FUNCTION_BLOCK ClearLinkEIP
VAR_INPUT
	bEnable : BOOL;
END_VAR
VAR_OUTPUT
	pulse AT %Q* : INT; //num pulses
	outputRegister AT %Q* : INT;
	brakeRelease AT %Q* : BOOL;
	
	A : BOOL; //direction (F = inwards, T = outwards)
	B : BOOL; //home bit
	clear : BOOL;
	
	contact AT %I* : BOOL;
	home AT %I* : BOOL;
	outerLimit AT %I* : BOOL;
	innerLimit AT %I* : BOOL;
	
	hlfb AT %I* : REAL; //high level feedback, if -9999 then servo is idle
	
	homeSet : BOOL;
	busy : BOOL;
	error : BOOL;
	
	position : LREAL;
	targetPos : LREAL;
END_VAR
VAR
	pulseRequest : INT;
	pulser : TON;
	
	minHoming : TON;
	resetPulse : TP;
	
	step : Homing;
	mode : (DISABLE, HOLD, TARGET, CONTINUOUS, RESET_ERR);
END_VAR
VAR_STAT CONSTANT
	resetTime : TIME := T#1000MS;
	pulseWidth : TIME := T#40MS;
	pulseSeparation : TIME := T#40MS;
	unitsPerPulse : INT := 800; //800 Teknic units per revolution
	distancePerPulse : INT := 5; //5mm per revolution
END_VAR

//M-connector output register
outputRegister.0 := bEnable; 	//enable
outputRegister.1 := A; 			//direction bit
outputRegister.2 := B; 			//homing bit - set to TRUE on startup to begin homing, then set to FALSE to finish homing
outputRegister.3 := clear; 		//reset bit

resetPulse(IN:= , PT:= resetTime, Q=> clear, ET=> ); //reset timer

IF NOT bEnable THEN
	homeSet := FALSE;
	mode := HOLD;
END_IF

//set the bool outputs, all are listed for readability
homeSet := homeSet;
busy := hlfb <> -9999;
error := error;

override(); //if sensor limits are reached, this method blocks motion that would exceed the limits

CASE mode OF		
	HOLD: //hold current position, no motion
		pulse := 0;
		pulseRequest := 0;
	
	TARGET:	//target a given position
		IF WithinTolerance(position, targetPos, distancePerPulse) THEN
			pulseRequest := 0;
			mode := HOLD;
			
		ELSIF NOT busy THEN
			A :=  position < targetPos;
			(*
			2 options to traverse to a target position:
				a)  send all pulses at once - single continuous motion but may exceed limits
				b)  1 pulse at a time - choppy but safer
			*)
			pulseRequest := TO_INT(ABS(position - targetPos)/distancePerPulse);
			//pulseRequest := 1;
			
		END_IF
		
	CONTINUOUS: //single pulses in the direction specified by moveContinuous()
		pulseRequest := 1;
		
	RESET_ERR: //reset pulse
		pulse := 0;
		pulseRequest := 0;
		
		resetPulse.IN := TRUE;
		mode := HOLD;
		(*
		IF resetTimer.Q THEN
			resetTimer.IN := FALSE;
			mode := HOLD;
		END_IF
		*)
		
END_CASE

sequence();

METHOD homingSequence : BOOL
minHoming(IN:= , PT:= T#1S, Q=> , ET=> ); //IN and OUT should be held for at least 1 second - may be removed for deployment

IF NOT bEnable THEN //homing does not begin until software enable
	RETURN;
END_IF

CASE step OF
	Homing.IDLE:
		bEnable := FALSE;
		A := FALSE;
		B := FALSE;
		brakeRelease := TRUE;
		
		homeSet := FALSE;
		step := Homing.IN;
		
	Homing.IN: //let insertion drop to inner limit before homing
		bEnable := FALSE;
		A := FALSE;
		B := FALSE;
		brakeRelease := TRUE;
		
		minHoming.IN := TRUE;
		
		IF NOT innerLimit AND minHoming.Q THEN
			minHoming.IN := FALSE;
			step := Homing.OUT;
		END_IF
	
	Homing.OUT: //home to outer limit
		bEnable := TRUE;
		A := FALSE;
		B := TRUE;
		brakeRelease := TRUE;
		
		minHoming.IN := TRUE;
		
		IF NOT home AND minHoming.Q THEN
			minHoming.IN := FALSE;
			step := Homing.DONE;
		END_IF
		
	Homing.DONE: //set home
		bEnable := TRUE;
		A := FALSE;
		B := FALSE;
		brakeRelease := TRUE;
		
		position := 0;
		
		homeSet := TRUE;
		homingSequence := TRUE;
		
		mode := HOLD;
		step := Homing.IDLE;
		
END_CASE
END_METHOD

METHOD moveAbsolute : BOOL
VAR_INPUT
	newTarget : LREAL;
END_VAR
targetPos := newTarget;
mode := TARGET;
END_METHOD

METHOD moveContinuous : BOOL
VAR_INPUT
	direction : MC_Direction;
END_VAR
IF direction = MC_Negative_Direction THEN
	A := FALSE;
ELSIF direction = MC_Positive_Direction THEN
	A := TRUE;
END_IF

mode := CONTINUOUS;
END_METHOD

METHOD PRIVATE override : BOOL
VAR_INPUT
END_VAR
(*
IF (*NOT*) home THEN //block outwards motion
	position := 0;
	IF A THEN
		mode := HOLD;
	END_IF
	
ELSIF (*NOT*) outerLimit AND_THEN A THEN //block outwards motion
	mode := HOLD;

ELSIF (*NOT*) innerLimit AND_THEN NOT A THEN //block inwards motion
	mode := HOLD;
	
END_IF
*)


IF
	((*NOT*) home AND_THEN A) OR
	((*NOT*) outerLimit AND_THEN A) OR
	((*NOT*) innerLimit AND_THEN NOT A)
THEN
	mode := HOLD;
END_IF


IF (*NOT*) home THEN //block outwards motion
	position := 0;
END_IF
END_METHOD

METHOD reset : BOOL
VAR_INPUT
END_VAR
mode := RESET_ERR;
END_METHOD

METHOD PRIVATE sequence : BOOL
VAR_INPUT
END_VAR
IF hlfb > -9999 THEN //servo is active
	IF A THEN //positive direction
		position := position + (distancePerPulse * pulse);
	ELSE //negative direction
		position := position - (distancePerPulse * pulse);
	END_IF
	pulse := 0; //pulses already received, can be set to 0 so position change is not compounded

ELSIF pulse = 0 THEN //servo is not active
	pulse := pulseRequest;
	pulseRequest := 0; //remove this if not working as intended
	
END_IF
END_METHOD

METHOD stop : BOOL
VAR_INPUT
END_VAR
mode := HOLD;
END_METHOD

END_FUNCTION_BLOCK

(* stored: Version 1.1.0.1, ProductVersion 3.1.4024.11
   POU ClearLinkEIP: Id {82d395c8-897a-4c3b-989f-b99dc8146760}, SpecialFunc None
   Folder Private: Id {5799debc-a080-4517-ac59-8af37dba3ca0}
   Method homingSequence: Id {ed7f9015-f217-4688-b191-db86d43e2b15}
   Method moveAbsolute: Id {dc77def1-bef9-43df-afd0-8ca352bd4ae2}
   Method moveContinuous: Id {56e37924-ed1f-434c-b8b5-86f83bcd5e14}
   Method override: Id {12f80332-3269-42b5-a267-e03e0f51e546}
   Method reset: Id {b78ab13d-678d-4b52-8830-ac5e90a85d68}
   Method sequence: Id {d3e76146-deb6-4a1c-bf00-057dae828590}
   Method stop: Id {b371037c-73c2-41cf-af60-cf703d5e079a} *)
